PROGRAM PRG_MasterCycle
VAR
	
		tonCaseTimDelay    	: ARRAY [1..20] OF Tc2_Standard.TON;
	    rtrigCaseTriger    	: ARRAY [1..10] OF Tc2_Standard.R_TRIG;
		ftrigCaseTriger		: ARRAY [1..10] OF Tc2_Standard.F_TRIG;
	   	rtrigFaultMachine  	: Tc2_Standard.R_TRIG;	
		
		biClamp				: BOOL;
		biPartPresent		: BOOL;
		


		bAutoCycleStop		: BOOL;
		
		bCycleFlag			: BOOL;
		bGreenLED			: BOOL;
		bRedLED				: BOOL;
		bEndCycleFlag		: BOOL;
		bStationsStopped	: BOOL;
		bHeighTestCompleteFlag : BOOL;
		bLeakTestCompleteFlag : BOOL;
		i					: DINT;
		
		


END_VAR
VAR_IN_OUT
	stStationStruct          : ST_StandardStationStruct;
END_VAR

ACT_LinkIO();
ACT_TimTrig();
stStationStruct.bStationInProgress := stStationStruct.nState>=1100 AND stStationStruct.nState<=1600;

IF stStationStruct.nState <700 OR  stStationStruct.nState > 4000 THEN
	GVL_HMI_GLOBAL.sActualProcess := ""; 
	GVL_MASTER.stNest.bPiecePass 	:= FALSE;
	GVL_MASTER.stNest.bPieceReject 	:= FALSE;
	bGreenLED						:= FALSE;
	bRedLED							:= FALSE;
	GVL_MASTER.stNest.bHeightPass 	:= FALSE;
	GVL_MASTER.stNest.bLeakPass 	:= FALSE;
	GVL_MASTER.stNest.bVisionPass 	:= FALSE;
	GVL_MASTER.stNest.bHeightReject := FALSE;
	GVL_MASTER.stNest.bLeakReject	:= FALSE;
	GVL_MASTER.stNest.bVisionReject := FALSE;
END_IF

IF rtrigCaseTriger[3].Q THEN
GVL_PERSIST.stPartsInspection.nPartsGood:= GVL_PERSIST.stPartsInspection.nPartsGood +1;
GVL_PERSIST.stPartsInspection.nTotalPartsGood := GVL_PERSIST.stPartsInspection.nTotalPartsGood+1;
ELSIF GVL_HMI_GLOBAL.bResetGoodParts THEN
GVL_PERSIST.stPartsInspection.nPartsGood:=0;	
END_IF


IF rtrigCaseTriger[4].Q THEN
	GVL_PERSIST.stPartsInspection.nPartsFailed:=GVL_PERSIST.stPartsInspection.nPartsFailed+1;
	GVL_PERSIST.stPartsInspection.nTotalPartsFailed:= GVL_PERSIST.stPartsInspection.nTotalPartsFailed+1;
ELSIF GVL_HMI_GLOBAL.bResetFailedParts THEN
	GVL_PERSIST.stPartsInspection.nPartsFailed:=0;
END_IF

IF stStationStruct.nState < 700 THEN
	 GVL_HMI_GLOBAL.sMessageToOperator := "Press Reset Button to Home Machine";
END_IF

CASE stStationStruct.nState OF
	
100: 
   bAutoCycleStop := FALSE;
IF NOT GVL_MASTER.stMachineStatus.bSystemPowerUp THEN
	stStationStruct.nState := 200;
END_IF
200:
IF GVL_MASTER.stMachineStatus.bSystemInitialising THEN
	stStationStruct.nState := 300;
END_IF
300:
   GVL_Master.stStationSruct[1].bStationInitRequest := TRUE;
   GVL_Master.stStationSruct[2].bStationInitRequest := TRUE;
   GVL_Master.stStationSruct[3].bStationInitRequest := TRUE;
   
IF GVL_Master.stStationSruct[1].bStationInitRequest AND GVL_Master.stStationSruct[2].bStationInitRequest AND
   GVL_Master.stStationSruct[3].bStationInitRequest  THEN
	stStationStruct.nState := 400;
END_IF
400:
IF NOT GVL_Master.stStationSruct[1].bStationInitRequest AND NOT GVL_Master.stStationSruct[2].bStationInitRequest AND
   NOT GVL_Master.stStationSruct[3].bStationInitRequest THEN
	stStationStruct.nState := 500;   
END_IF 
500:
   GVL_Master.stStationSruct[1].bStationAcknowledge := TRUE;
   GVL_Master.stStationSruct[2].bStationAcknowledge := TRUE;
   GVL_Master.stStationSruct[3].bStationAcknowledge := TRUE;
IF   GVL_Master.stStationSruct[1].bStationAcknowledge AND  GVL_Master.stStationSruct[2].bStationAcknowledge AND
     GVL_Master.stStationSruct[3].bStationAcknowledge THEN
     stStationStruct.nState := 600;
END_IF
600:
IF GVL_Master.stStationSruct[1].bStationHomed AND GVL_Master.stStationSruct[2].bStationHomed AND GVL_Master.stStationSruct[3].bStationHomed  THEN
   GVL_Master.stStationSruct[1].bStationAcknowledge := FALSE;
   GVL_Master.stStationSruct[2].bStationAcknowledge := FALSE;
   GVL_Master.stStationSruct[3].bStationAcknowledge := FALSE;
   stStationStruct.nState := 700;
END_IF
700: // All Station Homed and waiting for Autocycle 
   bAutoCycleStop := FALSE;
   GVL_HMI_GLOBAL.sActualProcess := "Waiting for Autocycle";
   IF GVL_MASTER.stMachineStatus.bSystemReadyToStart THEN 
	  GVL_HMI_GLOBAL.sMessageToOperator := "Press Start Button to Autocycle";
   ELSE GVL_HMI_GLOBAL.sMessageToOperator := "Press Reset Button to Reset machine";
   END_IF
   
IF GVL_Master.stMachineStatus.bSystemAutoCycle THEN
	stStationStruct.nState := 800;
ELSIF GVL_Master.stMachineStatus.bManualMode THEN
      stStationStruct.nState := 4000;
ELSIF GVL_Master.stMachineStatus.bSystemStopping AND NOT bStationsStopped  THEN
      stStationStruct.nState := 5000;
ELSIF GVL_Master.stMachineStatus.bCycleStopFault OR GVL_Master.stMachineStatus.bImmediateFault THEN
      stStationStruct.nState := 6000;	  
END_IF

IF tonCaseTimDelay[9].Q THEN
	stStationStruct.nState := 1000;
END_IF
800:
stStationStruct.nState := 1000;
1000: // System Autocycle

IF biPartPresent THEN
	GVL_HMI_GLOBAL.sMessageToOperator := "Remove Nest";
ELSE GVL_HMI_GLOBAL.sMessageToOperator := "Insert Nest to begin process";
END_IF


IF  rtrigCaseTriger [5].Q  AND NOT bEndCycleFlag THEN
	GVL_MASTER.stNest.bHeightPass 	:= FALSE;
	GVL_MASTER.stNest.bLeakPass 	:= FALSE;
	GVL_MASTER.stNest.bVisionPass 	:= FALSE;
	GVL_MASTER.stNest.bHeightReject := FALSE;
	GVL_MASTER.stNest.bLeakReject	:= FALSE;
	GVL_MASTER.stNest.bVisionReject := FALSE;
	GVL_MASTER.stNest.bPiecePass 	:= FALSE;
	GVL_MASTER.stNest.bPieceReject 	:= FALSE;
	GVL_MASTER.stNest.bNestPartProced := FALSE;
	GVL_MASTER.stNest.sHeightHMI 	:= "";
	GVL_MASTER.stNest.sLeakHMI 		:= "";
	GVL_MASTER.stNest.sVisionHMI 	:= "";
	GVL_MASTER.stNest.sPieceHMI 	:= "";
	bCycleFlag						:= TRUE;
	GVL_HMI_GLOBAL.sMessageToOperator := "Process in progress";
	GVL_HMI_GLOBAL.bResetPassAndFail:= TRUE;
	GVL_HMI_GLOBAL.sActualProcess := "";
	bGreenLED						:= FALSE;
	bRedLED							:= FALSE;
	GVL_HMI_GLOBAL.bRejectPieceAcknowledge := FALSE;
	stStationStruct.nState 			:= 1130;
	
ELSIF GVL_Master.stMachineStatus.bSystemStopping  THEN
      stStationStruct.nState := 5000;
ELSIF tonCaseTimDelay[10].Q THEN
	  bAutoCycleStop := TRUE;
      stStationStruct.nState := 5000;	
END_IF
1130:
IF tonCaseTimDelay[13].Q THEN
	GVL_HMI_GLOBAL.bResetPassAndFail:= FALSE;
	stStationStruct.nState 			:= 1132;
END_IF


//Vision Test
1132: 
	GVL_MASTER.anValueBeforeMeasurement := GVL_MASTER.aSensorCurrentValue;
	GVL_HMI_GLOBAL.sActualProcess := "Vision process"; 
	GVL_Master.stStationSruct[3].bStationRequest := TRUE;
	stStationStruct.nState := 1134;
1134:
IF GVL_Master.stStationSruct[3].bStationInProgress THEN
	stStationStruct.nState := 1136;
END_IF
1136:
IF GVL_Master.stStationSruct[3].bStationComplete AND NOT GVL_Master.stMachineStatus.bSystemStopping THEN
	stStationStruct.nState := 1138;
ELSIF GVL_Master.stMachineStatus.bSystemStopping OR ftrigCaseTriger [1].Q THEN
	stStationStruct.nState := 5000;
END_IF
1138:
GVL_HMI_GLOBAL.sMessageToOperator := "Toggle Clamp to continue the process";
IF rtrigCaseTriger [1].Q  THEN
	stStationStruct.nState := 1142;
ELSIF GVL_Master.stMachineStatus.bSystemStopping  THEN
      stStationStruct.nState := 5000;
ELSIF tonCaseTimDelay[10].Q THEN
	  bAutoCycleStop := TRUE;
      stStationStruct.nState := 5000;	

END_IF
//Leak test
1142: 
	GVL_HMI_GLOBAL.sMessageToOperator := "Process in progress";
	GVL_HMI_GLOBAL.sActualProcess := "Leak And Height test process"; 
	GVL_Master.stStationSruct[2].bStationRequest := TRUE;
	GVL_Master.stStationSruct[1].bStationRequest := TRUE;
	stStationStruct.nState := 1144;
1144:
IF GVL_Master.stStationSruct[2].bStationInProgress AND GVL_Master.stStationSruct[1].bStationInProgress THEN
	stStationStruct.nState := 1146;
END_IF
1146:
IF GVL_Master.stStationSruct[2].bStationComplete THEN
	bHeighTestCompleteFlag := TRUE;
END_IF
IF GVL_Master.stStationSruct[1].bStationComplete THEN
	bLeakTestCompleteFlag := TRUE;
END_IF

IF bHeighTestCompleteFlag AND bLeakTestCompleteFlag AND NOT GVL_Master.stMachineStatus.bSystemStopping THEN
	stStationStruct.nState := 1152;
	GVL_MASTER.bHeightTestacknowledge := TRUE;
ELSIF GVL_Master.stMachineStatus.bSystemStopping THEN
	stStationStruct.nState := 5000;
END_IF

1152: 
	GVL_MASTER.stNest.bNestPartProced 	:= TRUE;
	bHeighTestCompleteFlag				:= FALSE;
	bLeakTestCompleteFlag				:= FALSE;
IF tonCaseTimDelay[12].Q THEN
	GVL_MASTER.bHeightTestacknowledge := FALSE;
	stStationStruct.nState := 1220;
END_IF
	
1220:
IF GVL_MASTER.stNest.bHeightPass AND GVL_MASTER.stNest.bLeakPass AND GVL_MASTER.stNest.bVisionPass THEN
	GVL_MASTER.stNest.bPiecePass 	:= TRUE;
	GVL_MASTER.stNest.bPieceReject 	:= FALSE;
	GVL_MASTER.stNest.sPieceHMI 	:= "Pass";
	bGreenLED						:= TRUE;
	bRedLED							:= FALSE;
ELSE GVL_MASTER.stNest.bNestPartOK := FALSE;
	GVL_MASTER.stNest.sPieceHMI 	:= "Fail";
	GVL_MASTER.stNest.bPiecePass 	:= FALSE;
	GVL_MASTER.stNest.bPieceReject 	:= TRUE;
	bGreenLED						:= FALSE;
	bRedLED							:= TRUE;
END_IF
GVL_MASTER.stNest.sDate := GVL_HMI_GLOBAL.sSystemDate;
GVL_MASTER.stNest.sTime := GVL_HMI_GLOBAL.sSystemTime;

IF rtrigCaseTriger [8].Q THEN	
	
	FOR i :=200 TO 1 BY (-1) DO
		GVL_HMI_GLOBAL.aStatistics[i]	:= GVL_HMI_GLOBAL.aStatistics[i-1];
	END_FOR
	
	GVL_HMI_GLOBAL.aStatistics[1] := GVL_MASTER.stNest;
END_IF

IF tonCaseTimDelay[11].Q THEN
	stStationStruct.nState := 1500;
END_IF

1500:
IF GVL_Master.stStationSruct[1].bStationNotMoving AND GVL_Master.stStationSruct[2].bStationNotMoving AND GVL_Master.stStationSruct[3].bStationNotMoving THEN
	stStationStruct.nState := 1550;
END_IF
1550:
IF  GVL_MASTER.stNest.bPiecePass THEN	
	stStationStruct.nState := 1600;
ELSIF  GVL_MASTER.stNest.bPieceReject AND GVL_HMI_GLOBAL.bRejectPieceAcknowledge THEN
	stStationStruct.nState := 1600;
END_IF

1600:
GVL_HMI_GLOBAL.sMessageToOperator 				:= "Cycle Complete";   // **LAA 17092025
bEndCycleFlag	:= TRUE;
IF NOT GVL_MASTER.stMachineStatus.bSystemStopping  THEN 
	stStationStruct.nState := 1700;
ELSE 
    stStationStruct.nState := 5000;	
END_IF
1700:
GVL_HMI_GLOBAL.sMessageToOperator 				:= "Release Clamp";    // **LAA 17092025
IF rtrigCaseTriger [7].Q  THEN 
	stStationStruct.nState := 1000; 
END_IF

4000: 
IF NOT GVL_MASTER.stMachineStatus.bManualMode THEN
	stStationStruct.nState := 700;	
ELSIF GVL_MASTER.stMachineStatus.bCycleStopFault OR GVL_MASTER.stMachineStatus.bImmediateFault THEN
      stStationStruct.nState := 6000;		
END_IF

//stopping
5000:
	GVL_Master.stStationSruct[1].bNoCycleStopRequest := FALSE;
    GVL_Master.stStationSruct[2].bNoCycleStopRequest := FALSE;
	GVL_Master.stStationSruct[3].bNoCycleStopRequest := FALSE;
	

IF tonCaseTimDelay[6].Q AND (GVL_Master.stStationSruct[1].nState = 1000) AND (GVL_Master.stStationSruct[2].nState = 1000) 
                        AND (GVL_Master.stStationSruct[3].nState = 1000) THEN
	bAutoCycleStop := FALSE;
	
	stStationStruct.nState := 700;

	
END_IF

6000:
IF tonCaseTimDelay[1].Q THEN
	GVL_Master.stStationSruct[1].bStationInitRequest := FALSE;
	GVL_Master.stStationSruct[2].bStationInitRequest := FALSE;
	GVL_Master.stStationSruct[3].bStationInitRequest := FALSE;
	GVL_Master.stStationSruct[1].bStationRequest := FALSE;
	GVL_Master.stStationSruct[2].bStationRequest := FALSE;
    GVL_Master.stStationSruct[3].bStationRequest := FALSE;
	GVL_Master.stStationSruct[1].bStationAbort := TRUE;
    GVL_Master.stStationSruct[2].bStationAbort := TRUE;
	GVL_Master.stStationSruct[3].bStationAbort := TRUE;
	stStationStruct.nState := 100;
END_IF


END_CASE

//++++++++++++++++++++++++++++++++++++++++++++++++++++++++++++++++++++++++++++++++++++++++++++++++++++++++++++++++++++++++++++++++++++++

IF rtrigFaultMachine.Q THEN
   stStationStruct.nState := 6000;	  
END_IF

IF  (stStationStruct.nState = 4000) OR (stStationStruct.nState = 5000) OR (stStationStruct.nState = 6000) THEN
   GVL_Master.stStationSruct[1].bStationAcknowledge := FALSE;
   GVL_Master.stStationSruct[2].bStationAcknowledge := FALSE;
   GVL_Master.stStationSruct[3].bStationAcknowledge := FALSE;
   GVL_Master.stStationSruct[1].bStationInitRequest := FALSE;
   GVL_Master.stStationSruct[2].bStationInitRequest := FALSE;
   GVL_Master.stStationSruct[3].bStationInitRequest := FALSE;
END_IF

ACTION ACT_LinkIO:
// Initialisation Progres
IF GVL_Master.stStationSruct[1].bStationInProgressInit THEN
	GVL_Master.stStationSruct[1].bStationInitRequest := FALSE;
END_IF
IF GVL_Master.stStationSruct[2].bStationInProgressInit THEN
	GVL_Master.stStationSruct[2].bStationInitRequest := FALSE;
END_IF
IF GVL_Master.stStationSruct[3].bStationInProgressInit THEN
	GVL_Master.stStationSruct[3].bStationInitRequest := FALSE;
END_IF

// Cycle Progres
IF GVL_Master.stStationSruct[1].bStationInProgress THEN
	GVL_Master.stStationSruct[1].bStationRequest := FALSE;
END_IF
IF GVL_Master.stStationSruct[2].bStationInProgress THEN
	GVL_Master.stStationSruct[2].bStationRequest := FALSE;
END_IF
IF GVL_Master.stStationSruct[3].bStationInProgress THEN
	GVL_Master.stStationSruct[3].bStationRequest := FALSE;
END_IF

// Abort Station
IF GVL_Master.stStationSruct[1].nState = 100 THEN
	GVL_Master.stStationSruct[1].bStationAbort := FALSE;
END_IF
IF GVL_Master.stStationSruct[2].nState = 100 THEN	
    GVL_Master.stStationSruct[2].bStationAbort := FALSE;
END_IF	
IF GVL_Master.stStationSruct[3].nState = 100 THEN
	GVL_Master.stStationSruct[3].bStationAbort := FALSE;
END_IF

IF (GVL_Master.stStationSruct[1].nState = 100) OR (GVL_Master.stStationSruct[1].nState = 1000) THEN
	GVL_Master.stStationSruct[1].bNoCycleStopRequest := TRUE;
END_IF
IF (GVL_Master.stStationSruct[2].nState = 100) OR (GVL_Master.stStationSruct[2].nState = 1000) THEN	
    GVL_Master.stStationSruct[2].bNoCycleStopRequest := TRUE;
END_IF
IF (GVL_Master.stStationSruct[3].nState = 100) OR (GVL_Master.stStationSruct[3].nState = 1000) THEN	
	GVL_Master.stStationSruct[3].bNoCycleStopRequest := TRUE;
END_IF

IF  (GVL_Master.stStationSruct[1].nState = 1000) AND (GVL_Master.stStationSruct[2].nState = 1000) 
                        AND (GVL_Master.stStationSruct[3].nState = 1000) THEN
	bStationsStopped := TRUE;
ELSE bStationsStopped := FALSE;

END_IF

GVL_MASTER.stMasterControl.bAllStationsCycledStopped := (GVL_Master.stStationSruct[1].nState = 1000) AND (GVL_Master.stStationSruct[2].nState = 1000) 
                                         AND (GVL_Master.stStationSruct[3].nState = 1000)
										 AND  stStationStruct.nState=700;
										 
	biClamp									:= GVL_IO.dw_T02_EL1809.iCalmpClosed;
	biPartPresent							:=  GVL_IO.dw_T02_EL1809.iPartPresent;
	GVL_MASTER.stNest.bNestPresent			:= GVL_IO.dw_T02_EL1809.iCalmpClosed;
	GVL_IO.dw_T03_EL2809.qPassIndicatorGreen:= bGreenLED;
	GVL_IO.dw_T03_EL2809.qRejectIndicatorRed:= bRedLED;
	
IF ftrigCaseTriger[1].Q THEN
	bEndCycleFlag							:= FALSE;
END_IF
	
GVL_MASTER.aSensorCurrentValue[1] 					:= GVL_IO.dw_B08_DL_PN1.gt2_1_1CurrentValue;
GVL_MASTER.aSensorCurrentValue[2] 					:= GVL_IO.dw_B08_DL_PN1.gt2_1_2CurrentValue;
GVL_MASTER.aSensorCurrentValue[3] 					:= GVL_IO.dw_B08_DL_PN1.gt2_1_3CurrentValue;
GVL_MASTER.aSensorCurrentValue[4] 					:= GVL_IO.dw_B08_DL_PN1.gt2_2CurrentValue;
END_ACTION

ACTION ACT_TimTrig:
tonCaseTimDelay[1](IN:= (stStationStruct.nState = 6000),PT:=T#100MS); //
tonCaseTimDelay[2](IN:= (stStationStruct.nState = 5000),PT:=T#100MS); //
tonCaseTimDelay[3](IN:= (stStationStruct.nState = 1100),PT:=T#40MS);  //
tonCaseTimDelay[4](IN:= (stStationStruct.nState = 1140),PT:=T#250MS);
tonCaseTimDelay[5](IN:= (stStationStruct.nState = 1900),PT:=T#250MS);
tonCaseTimDelay[6](IN:= (stStationStruct.nState = 5000),PT:=T#250MS);
tonCaseTimDelay[7](IN:= (stStationStruct.nState = 1340),PT:=T#200MS);
tonCaseTimDelay[8](IN:= (stStationStruct.nState = 1320),PT:=T#500MS);
tonCaseTimDelay[9](IN:= (stStationStruct.nState = 800),PT:=T#3S);
tonCaseTimDelay[10](IN:= (stStationStruct.nState = 1000),PT:=T#10M);
tonCaseTimDelay[11](IN:= (stStationStruct.nState = 1220),PT:=T#1S);
tonCaseTimDelay[12](IN:= stStationStruct.nState = 1152,PT:=T#1S );
tonCaseTimDelay[13](IN:=(stStationStruct.nState = 1130),PT:=T#1S );
tonCaseTimDelay[14](IN:=,PT:=T#1S);
tonCaseTimDelay[15](IN:= );
tonCaseTimDelay[16](IN:= );
tonCaseTimDelay[17](IN:= );
tonCaseTimDelay[18](IN:= );
tonCaseTimDelay[19](IN:= );
tonCaseTimDelay[20](IN:= );

rtrigCaseTriger [1](CLK:= biClamp);
rtrigCaseTriger [2](CLK:= tonCaseTimDelay[2].Q);
rtrigCaseTriger [3](CLK:= GVL_MASTER.stNest.bPiecePass);
rtrigCaseTriger [4](CLK:= GVL_MASTER.stNest.bPieceReject);
rtrigCaseTriger [5](CLK:= biPartPresent );
rtrigCaseTriger [6](CLK:= );
rtrigCaseTriger [7](CLK:= NOT biClamp);  // **LAA 17092025);
rtrigCaseTriger [8](CLK:= );
rtrigCaseTriger [9](CLK:= );
rtrigCaseTriger [10](CLK:= );
rtrigFaultMachine(CLK:= GVL_MASTER.stMachineStatus.bCycleStopFault OR GVL_MASTER.stMachineStatus.bImmediateFault);

ftrigCaseTriger [1](CLK:= biPartPresent );
END_ACTION

END_PROGRAM

(* stored: Version 1.1.0.1, ProductVersion 3.1.4024.13
   POU PRG_MasterCycle: Id {b14bd733-545d-49f3-8554-8f69ba8d0550}, SpecialFunc None
   Action ACT_LinkIO: Id {06593384-a51e-4e83-9963-7bd33731aa41}
   Action ACT_TimTrig: Id {f0836fdf-c0d8-40ee-b7c7-a5b5ff4f0cd6} *)
